# B&R Automation Studio project lab2
Automation Studio 4.5.2.102

## Configuration Config2

CPU 4PP065.0571-P74, AutomationRuntime D4.52, Build 4.1.2, Safety 1.6

### Task classes (Cpu.sw)
```
Cyclic#4:
  Program <- Program.prg
Binaries: udbdef, TCData, iomap, ashwac, Role, sysconf, arconfig, asfw, User, ashwd
Libraries: DriveLib
```

### Hardware
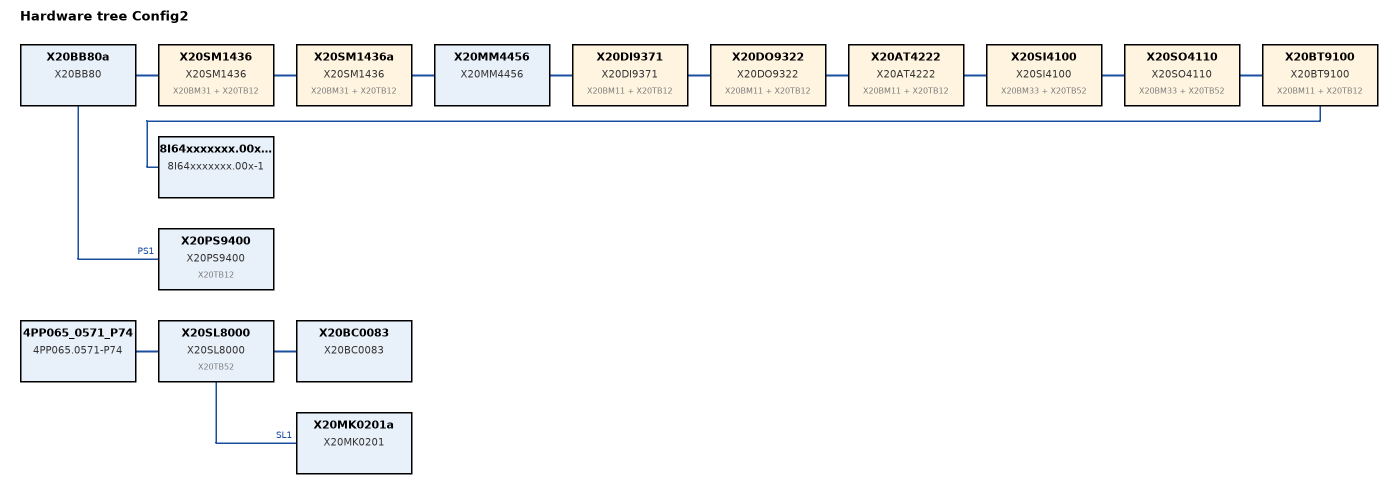
```
4PP065_0571_P74 : 4PP065.0571-P74 v1.1.2.0
  Connector IF5:
    ActivateDevice = 1
    Mode = Manual
    InternetAddress = 10.0.1.10
    SubnetMask = 255.255.255.0
  ConfigurationID = labBR
8I64xxxxxxx.00x-1 : 8I64xxxxxxx.00x-1 v1.3.9.1  [X2X1 -> X20BT9100.X2X1 [Cable Type=X2XCable, Length=10, Version=1.0.0.2]]
  FunctionModel = Standard
  packedETAD = packed
  packedETI = packed
  packedCMDD = packed
X20AT4222 : X20AT4222 v1.2.3.0  [SS1 -> X20TB12i.SS; SL -> X20BM11f.SL1]
X20BB80a : X20BB80 v1.0.2.0
X20BC0083 : X20BC0083 v2.7.0.0  [PLK1 -> X20SL8000.PLK2 (NodeNumber=2) [Cable Type=PowerlinkCable, Length=10, Version=1.0.0.2]; SL -> X20BB80a.SL1]
X20BM11 : X20BM11 v1.0.0.1  [X2X1 -> X20MM4456.X2X2]
X20BM11c : X20BM11 v1.0.0.1  [X2X1 -> X20BM11.X2X2]
X20BM11e : X20BM11 v1.0.0.1  [X2X1 -> X20BM33c.X2X2]
X20BM11f : X20BM11 v1.0.0.1  [X2X1 -> X20BM11c.X2X2]
X20BM31a : X20BM31 v1.0.0.1  [X2X1 -> X20BB80a.IF1]
X20BM31b : X20BM31 v1.0.0.1  [X2X1 -> X20BM31a.X2X2]
X20BM33 : X20BM33 v1.0.0.4  [X2X1 -> X20BM11f.X2X2]
X20BM33c : X20BM33 v1.0.0.4  [X2X1 -> X20BM33.X2X2]
X20BT9100 : X20BT9100 v1.0.3.0  [SS1 -> X20TB12h.SS; SL -> X20BM11e.SL1]
X20DI9371 : X20DI9371 v1.0.2.0  [SS1 -> X20TB12.SS; SL -> X20BM11.SL1]
X20DO9322 : X20DO9322 v1.0.3.0  [SS1 -> X20TB12f.SS; SL -> X20BM11c.SL1]
X20MK0201a : X20MK0201 v1.0.0.0  [SL -> X20SL8000.SL1]
X20MM4456 : X20MM4456 v1.1.5.0  [X2X1 -> X20BM31b.X2X2]
X20PS9400 : X20PS9400 v1.0.2.4  [SS1 -> X20TB12b.SS; PS -> X20BB80a.PS1]
X20SI4100 : X20SI4100 v1.10.1.1  [SS1 -> X20TB52.SS; SL -> X20BM33.SL1]
X20SL8000 : X20SL8000 v1.6.5.1  [PLK1 -> 4PP065_0571_P74.IF4 (NodeNumber=1) [Cable Type=PowerlinkCable, Length=10, Version=1.0.0.2]; PLK2 -> X20BC0083.PLK1 (NodeNumber=1) [Cable Type=PowerlinkCable, Length=10, Version=1.0.0.2]; SS1 -> X20TB52a.SS]
  SafeProject = SafeLOGIC-1
X20SM1436 : X20SM1436 v1.4.2.1  [SS1 -> X20TB12a.SS; SL -> X20BM31a.SL1]
X20SM1436a : X20SM1436 v1.4.2.1  [SS1 -> X20TB12c.SS; SL -> X20BM31b.SL1]
X20SO4110 : X20SO4110 v1.10.1.1  [SS1 -> X20TB52d.SS; SL -> X20BM33c.SL1]
  SafeModuleID = 3
X20TB12 : X20TB12 v1.0.0.0
X20TB12a : X20TB12 v1.0.0.0
X20TB12b : X20TB12 v1.0.0.0
X20TB12c : X20TB12 v1.0.0.0
X20TB12f : X20TB12 v1.0.0.0
X20TB12h : X20TB12 v1.0.0.0
X20TB12i : X20TB12 v1.0.0.0
X20TB52 : X20TB52 v1.0.0.1
X20TB52a : X20TB52 v1.0.0.1
X20TB52d : X20TB52 v1.0.0.1
```

### IoMap.iom - 4PP065_0571_P74/IoMap.iom
```iecst
VAR_CONFIG
	::Program:Door.speed AT %QW."8I64xxxxxxx.00x-1".LFRD_Output;
	::Program:Motor.state AT %IW."8I64xxxxxxx.00x-1".ETAD_Input;
	::Program:Motor.command AT %QW."8I64xxxxxxx.00x-1".CMDD_Output;
	::Program:Led.led1 AT %QX."X20DO9322".DigitalOutput02;
	::Program:Led.led2 AT %QX."X20DO9322".DigitalOutput03;
	::Program:Led.led3 AT %QX."X20DO9322".DigitalOutput04;
	::Program:Led.led4 AT %QX."X20DO9322".DigitalOutput05;
	::Program:Door.direction AT %IX."X20DI9371".DigitalInput01;
	::Program:Door.sw1 AT %IX."X20DI9371".DigitalInput02;
	::Program:Door.sw2 AT %IX."X20DI9371".DigitalInput03;
	::Program:Door.sw3 AT %IX."X20DI9371".DigitalInput04;
	::Program:Door.sw4 AT %IX."X20DI9371".DigitalInput05;
END_VAR
```

## Configuration Config3

### Task classes (Cpu.sw)
```
Cyclic#1:
  ncsdcctrl <- ncsdcctrl.prg
NcDataObjects: acp10etxen <- acp10etxen.dob, gAxis01a <- gAxis01obj.gAxis01a.dob, gAxis01i <- gAxis01obj.gAxis01i.dob
Libraries: Acp10man, Acp10par, NcGlobal, Acp10sdc, Acp10_MC, brsystem, sys_lib, runtime, AsBrStr
```

## Logical view

Binary libraries used (declarations not repeated): operator, astime, AsIecCon, runtime, Acp10man, Acp10par, NcGlobal, Acp10sdc, Acp10_MC, brsystem, sys_lib, AsBrStr

### Package Logical/Libraries - Global libraries

### Library Logical/Libraries/DriveLib (ANSIC)

#### Types.typ - Exported data types
```iecst
TYPE
	list_of_state :
		(
		STATE_SWITCHED_ON := 1,
		STATE_READY := 2
		);
	list_of_door :
		(
		ST_INIT := 1,
		ST_UNKNOWN := 2,
		ST_OPEN := 3,
		ST_DEC_NEG := 4,
		ST_DEC_POS := 5,
		ST_NEG := 6,
		ST_POS := 7,
		ST_ACC_NEG := 8,
		ST_ACC_POS := 9,
		ST_CLOSE := 10
		);
	list_of_command :
		(
		CMD_ENABLE := 1,
		CMD_SWITCH_ON := 2,
		CMD_SHUTDOWN := 3
		);
END_TYPE
```

#### DrivelIB.fun - Exported functions and function blocks
```iecst
{REDUND_ERROR} FUNCTION_BLOCK DriveStateMashine (*TODO: Add your comment here*) (*$GROUP=User,$CAT=User,$GROUPICON=User.png,$CATICON=User.png*)
	VAR_INPUT
		state : UINT;
		enable : BOOL;
		sta : UINT;
	END_VAR
	VAR_OUTPUT
		command : UINT;
		speed : INT;
		com : UINT;
	END_VAR
END_FUNCTION_BLOCK

{REDUND_ERROR} FUNCTION_BLOCK DoorStateMashine (*TODO: Add your comment here*) (*$GROUP=User,$CAT=User,$GROUPICON=User.png,$CATICON=User.png*)
	VAR_INPUT
		state : list_of_door;
		sw1 : BOOL;
		sw2 : BOOL;
		sw3 : BOOL;
		sw4 : BOOL;
		direction : BOOL;
	END_VAR
	VAR_OUTPUT
		speed : INT;
	END_VAR
	VAR
		led_state : LedStateMashine;
	END_VAR
END_FUNCTION_BLOCK

{REDUND_ERROR} FUNCTION_BLOCK LedStateMashine (*TODO: Add your comment here*) (*$GROUP=User,$CAT=User,$GROUPICON=User.png,$CATICON=User.png*)
	VAR_INPUT
		state : UINT;
	END_VAR
	VAR_OUTPUT
		led1 : BOOL;
		led2 : BOOL;
		led3 : BOOL;
		led4 : BOOL;
		timer : INT;
	END_VAR
END_FUNCTION_BLOCK
```

#### DriveStateMashine.c
```c
#include <bur/plctypes.h>
#ifdef __cplusplus
	extern "C"
	{
#endif
	#include "DriveLib.h"
#ifdef __cplusplus
	};
#endif
/* TODO: Add your comment here */
void DriveStateMashine(struct DriveStateMashine* inst)
{
	inst->command = CMD_SHUTDOWN;

	if (inst->enable == 0 || inst->state & 0x6F != STATE_SWITCHED_ON)
	{
		inst->command = CMD_SHUTDOWN;
	}
	else
	{
		if (inst->state & 0x6F != STATE_SWITCHED_ON)
		{
			inst->command = CMD_SWITCH_ON;
		}
		else
		{
			inst->command = CMD_ENABLE;
		}
	}
}
```

#### DoorStateMashine.c
```c
#include <bur/plctypes.h>
#ifdef __cplusplus
	extern "C"
	{
#endif
	#include "DriveLib.h"
#ifdef __cplusplus
	};
#endif
/* TODO: Add your comment here */
void DoorStateMashine(struct DoorStateMashine* inst)
{
	if (inst->state == ST_INIT)
	{inst->state = ST_UNKNOWN;
		inst->led_state.state=0000; LedStateMashine(&inst->led_state);
		inst->led_state.state=1111; LedStateMashine(&inst->led_state);
		inst->led_state.state=0000; LedStateMashine(&inst->led_state);
		return;
	}
	if (inst->state == ST_UNKNOWN)
	{
		if (inst->sw1 == 1 && inst->direction == 0)
		{inst->state = ST_OPEN;inst->led_state.state=0000; LedStateMashine(&inst->led_state); inst->speed = 0;}
		else if (inst->sw2 == 1 && inst->direction == 1)
		{inst->state = ST_CLOSE; inst->led_state.state=1111; LedStateMashine(&inst->led_state); inst->speed = 0;}
		return;
	}

	if (inst->state == ST_OPEN && inst->direction == 1)
	{inst->state = ST_ACC_POS; inst->led_state.state=1000; LedStateMashine(&inst->led_state); inst->speed = 10; return;}

	if (inst->state == ST_CLOSE && inst->direction == 0)
	{inst->state = ST_ACC_NEG; inst->led_state.state=1110; LedStateMashine(&inst->led_state); inst->speed = -10; return;}

	if (inst->state == ST_ACC_POS)
	{
		if (inst->direction == 1)
		{inst->state = ST_DEC_NEG; inst->led_state.state=1000; LedStateMashine(&inst->led_state); inst->speed = -10;}
		else if (inst->sw2 == 1)
		{inst->state = ST_POS; inst->led_state.state=1100; LedStateMashine(&inst->led_state); inst->speed = 100;}
		return;
	}

	if (inst->state == ST_ACC_NEG)
	{
		if (inst->direction == 0)
		{inst->state = ST_DEC_POS; inst->led_state.state=1110; LedStateMashine(&inst->led_state);inst->speed = 10; }
		else if (inst->sw3 == 1)
		{inst->state = ST_NEG; inst->led_state.state=1100; LedStateMashine(&inst->led_state); inst->speed = -100;}
		return;
	}

	if (inst->state == ST_POS)
	{
		if (inst->direction == 1)
		{inst->state = ST_NEG; inst->led_state.state=1100; LedStateMashine(&inst->led_state); inst->speed = -100;}
		else if (inst->sw3 == 1)
		{inst->state = ST_DEC_POS; inst->led_state.state=1110; LedStateMashine(&inst->led_state); inst->speed = 10;}
		return;
	}

	if (inst->state == ST_NEG)
	{
		if (inst->direction == 0)
		{inst->state = ST_POS; inst->led_state.state=1100; LedStateMashine(&inst->led_state); inst->speed = 100;}
		else if (inst->sw2 == 1)
		{inst->state = ST_DEC_NEG;inst->led_state.state=1000; LedStateMashine(&inst->led_state); inst->speed = -10;}
		return;
	}

	if (inst->state == ST_DEC_POS && inst->sw4 == 1)
	{inst->state = ST_CLOSE; inst->led_state.state=1111; LedStateMashine(&inst->led_state); inst->speed = 0; return;}

	if (inst->state == ST_DEC_NEG && inst->sw1 == 1)
	{inst->state = ST_OPEN; inst->led_state.state=0000; LedStateMashine(&inst->led_state); inst->speed = 0; return;}

}
```

#### LedStateMashine.c
```c
#include <bur/plctypes.h>
#ifdef __cplusplus
	extern "C"
	{
#endif
	#include "DriveLib.h"
#ifdef __cplusplus
	};
#endif+
/* TODO: Add your comment here */
void LedStateMashine(struct LedStateMashine* inst)
{
	if (inst->timer % 10 < 5)
	{
		inst->led1 = 0;
		inst->led2 = 0;
		inst->led3 = 0;
		inst->led4 = 0;
	}
	else
	{
		inst->led1 = inst->state & 0x00;
		inst->led2 = inst->state & 0x01;
		inst->led3 = inst->state & 0x02;
		inst->led4 = inst->state & 0x03;
	}
}
```

### Program Logical/Program (ANSIC)

#### Variables.var
```iecst
VAR
	Led : LedStateMashine;
	Door : DoorStateMashine;
	Motor : DriveStateMashine;
END_VAR
```

#### Cyclic.c
```c
#include <bur/plctypes.h>

#ifdef _DEFAULT_INCLUDES
	#include <AsDefault.h>
#endif

void _CYCLIC ProgramCyclic(void)
{
	DoorStateMashine(&Door);
	if (Door.sw1 || Door.sw4)
	{Motor.enable = 1;}
	else
	{Motor.enable = 0;}
	Motor.speed = Door.speed;
	DriveStateMashine(&Motor);

}
```

Listed in the project but not available here: Logical/Global.typ, Logical/Global.var, Logical/Libraries/DriveLib/Constants.var, Logical/ncsdcctrl, Logical/acp10etxen, Logical/gAxis01obj
